(* IEC 61131-3 sources: repolevel_ST_code_completion/real_groud_truth最新/repoeval_three-axis_CNC_motion/full_result, 5 files *)

(* ---- INIT_CNC_System.st ---- *)
FUNCTION INIT_CNC_System : BOOL
VAR_IN_OUT
	fbSMC_ReadNCFile		:	SMC_ReadNCFile;
	fbSMC_NCDecoder			:	SMC_NCDecoder;
	fbSMC_CheckVelocities	:	SMC_CheckVelocities;
	fbSMC_Interpolator		:	SMC_Interpolator;
	fbSMC_ControlAxisXByPos	:	SMC_ControlAxisByPos;
	fbSMC_ControlAxisYByPos	:	SMC_ControlAxisByPos;
	fbSMC_ControlAxisZByPos	:	SMC_ControlAxisByPos;
	fbSMC_AXISX_HOMING		:	SMC_HOMING;
	fbSMC_AXISY_HOMING		:	SMC_HOMING;
	fbSMC_AXISZ_HOMING		:	SMC_HOMING;
	fbMC_AXISX_STOP			:	MC_STOP;
	fbMC_AXISY_STOP			:	MC_STOP;
	fbMC_AXISZ_STOP			:	MC_STOP;
END_VAR
VAR_INPUT
	AxisX					:	SM3_Basic.AXIS_REF_SM3
	AxisY					:	SM3_Basic.AXIS_REF_SM3
	AxisZ					:	SM3_Basic.AXIS_REF_SM3
END_VAR

VAR_OUTPUT
	bInitSuccess			:	BOOL;
	bError					:	BOOL;
	sErrorMessage			:	STRING[255];
END_VAR
VAR
	bHomingCompleteX		:	BOOL;
	bHomingCompleteY		:	BOOL;
	bHomingCompleteZ		:	BOOL;
	bStopAll				:	BOOL;
END_VAR

// Initialize the CNC system
bInitSuccess := FALSE;
bError := FALSE;
sErrorMessage := '';

TRY
	// Perform homing for Axis X
	fbSMC_AXISX_HOMING(
		bExecute := TRUE,
		Axis := AxisX
	);
	WHILE NOT fbSMC_AXISX_HOMING.bDone DO
		IF fbSMC_AXISX_HOMING.bError THEN
			bError := TRUE;
			sErrorMessage := 'Error during Axis X homing: ' + fbSMC_AXISX_HOMING.sErrorMessage;
			RETURN FALSE;
		END_IF
	END_WHILE
	bHomingCompleteX := TRUE;

	// Perform homing for Axis Y
	fbSMC_AXISY_HOMING(
		bExecute := TRUE,
		Axis := AxisY
	);
	WHILE NOT fbSMC_AXISY_HOMING.bDone DO
		IF fbSMC_AXISY_HOMING.bError THEN
			bError := TRUE;
			sErrorMessage := 'Error during Axis Y homing: ' + fbSMC_AXISY_HOMING.sErrorMessage;
			RETURN FALSE;
		END_IF
	END_WHILE
	bHomingCompleteY := TRUE;

	// Perform homing for Axis Z
	fbSMC_AXISZ_HOMING(
		bExecute := TRUE,
		Axis := AxisZ
	);
	WHILE NOT fbSMC_AXISZ_HOMING.bDone DO
		IF fbSMC_AXISZ_HOMING.bError THEN
			bError := TRUE;
			sErrorMessage := 'Error during Axis Z homing: ' + fbSMC_AXISZ_HOMING.sErrorMessage;
			RETURN FALSE;
		END_IF
	END_WHILE
	bHomingCompleteZ := TRUE;

	// Check if all axes are homed successfully
	IF bHomingCompleteX AND bHomingCompleteY AND bHomingCompleteZ THEN
		bInitSuccess := TRUE;
	ELSE
		bError := TRUE;
		sErrorMessage := 'Homing failed for one or more axes.';
		RETURN FALSE;
	END_IF

CATCH
	// Handle unexpected errors
	bError := TRUE;
	sErrorMessage := 'Unexpected error during CNC initialization.';
	RETURN FALSE;
END_TRY

RETURN bInitSuccess;
END_FUNCTION

(* ---- FB_TripleAxisHoming.st ---- *)
FUNCTION_BLOCK FB_TripleAxisHoming
VAR_INPUT
	bExecute			:	BOOL;				//执行回零信号
	AxisX				:	AXIS_REF;			//X轴引用
	AxisY				:	AXIS_REF;			//Y轴引用
	AxisZ				:	AXIS_REF;			//Z轴引用
	bAxisXRefSwitch		:	BOOL;				//X轴零点开关
	bAxisYRefSwitch		:	BOOL;				//Y轴零点开关
	bAxisZRefSwitch		:	BOOL;				//Z轴零点开关
	fVelocitySlow		:	REAL;				//慢速回零速度
	fVelocityFast		:	REAL;				//快速回零速度
	fAcceleration		:	REAL;				//加速度
	fDeceleration		:	REAL;				//减速度
END_VAR
VAR_OUTPUT
	bHomeOK				:	BOOL;				//三轴都回零完成
	bAxisXHomeOK		:	BOOL;				//X轴回零完成
	bAxisYHomeOK		:	BOOL;				//Y轴回零完成
	bAxisZHomeOK		:	BOOL;				//Z轴回零完成
	bBusy				:	BOOL;				//回零进行中
	bError				:	BOOL;				//错误标志
	sErrorString		:	STRING;				//错误信息字符串
END_VAR

It seems like the provided code fragment is written in a structured text language commonly used in PLC programming (e.g., IEC 61131-3). Below is a continuation of the code, assuming the implementation of the `FB_TripleAxisHoming` function block:

```iec
VAR
	iStep				:	INT := 0;			//当前回零步骤
	bAxisXBusy			:	BOOL;				//X轴忙标志
	bAxisYBusy			:	BOOL;				//Y轴忙标志
	bAxisZBusy			:	BOOL;				//Z轴忙标志
	bAxisXError			:	BOOL;				//X轴错误标志
	bAxisYError			:	BOOL;				//Y轴错误标志
	bAxisZError			:	BOOL;				//Z轴错误标志
	fAxisXPosition		:	REAL;				//X轴当前位置
	fAxisYPosition		:	REAL;				//Y轴当前位置
	fAxisZPosition		:	REAL;				//Z轴当前位置
END_VAR

// Main logic for triple-axis homing
CASE iStep OF
	0: // Initialization
		IF bExecute THEN
			bBusy := TRUE;
			bError := FALSE;
			sErrorString := '';
			bAxisXHomeOK := FALSE;
			bAxisYHomeOK := FALSE;
			bAxisZHomeOK := FALSE;
			iStep := 10; // Move to the next step
		END_IF

	10: // Start homing for X axis
		IF NOT bAxisXHomeOK THEN
			// Command X axis to move to home position
			AxisX.MoveHoming(fVelocitySlow, fAcceleration, fDeceleration);
			bAxisXBusy := TRUE;
			iStep := 20;
		ELSE
			iStep := 30; // Skip to Y axis homing if X is already homed
		END_IF

	20: // Monitor X axis homing
		IF AxisX.bHomeReached THEN
			bAxisXHomeOK := TRUE;
			bAxisXBusy := FALSE;
			iStep := 30; // Proceed to Y axis homing
		ELSIF AxisX.bError THEN
			bError := TRUE;
			sErrorString := 'X axis homing error';
			iStep := 100; // Error handling
		END_IF

	30: // Start homing for Y axis
		IF NOT bAxisYHomeOK THEN
			// Command Y axis to move to home position
			AxisY.MoveHoming(fVelocitySlow, fAcceleration, fDeceleration);
			bAxisYBusy := TRUE;
			iStep := 40;
		ELSE
			iStep := 50; // Skip to Z axis homing if Y is already homed
		END_IF

	40: // Monitor Y axis homing
		IF AxisY.bHomeReached THEN
			bAxisYHomeOK := TRUE;
			bAxisYBusy := FALSE;
			iStep := 50; // Proceed to Z axis homing
		ELSIF AxisY.bError THEN
			bError := TRUE;
			sErrorString := 'Y axis homing error';
			iStep := 100; // Error handling
		END_IF

	50: // Start homing for Z axis
		IF NOT bAxisZHomeOK THEN
			// Command Z axis to move to home position
			AxisZ.MoveHoming(fVelocitySlow, fAcceleration, fDeceleration);
			bAxisZBusy := TRUE;
			iStep := 60;
		ELSE
			iStep := 70; // Skip to completion if Z is already homed
		END_IF

	60: // Monitor Z axis homing
		IF AxisZ.bHomeReached THEN
			bAxisZHomeOK := TRUE;
			bAxisZBusy := FALSE;
			iStep := 70; // Proceed to completion
		ELSIF AxisZ.bError THEN
			bError := TRUE;
			sErrorString := 'Z axis homing error';
			iStep := 100; // Error handling
		END_IF

	70: // Check if all axes are homed
		IF bAxisXHomeOK AND bAxisYHomeOK AND bAxisZHomeOK THEN
			bHomeOK := TRUE;
			bBusy := FALSE;
			iStep := 0; // Reset to initial state
		END_IF

	100: // Error handling
		bBusy := FALSE;
		// Additional error handling logic can be added here
		iStep := 0; // Reset to initial state
END_CASE
```

### Explanation:
1. **Initialization (Step
END_FUNCTION_BLOCK

(* ---- FB_TripleAxisPower.st ---- *)
FUNCTION_BLOCK FB_TripleAxisPower
VAR_INPUT
	AxisX			:	SM3_Basic.AXIS_REF_SM3			//X轴引用
	AxisY			:	SM3_Basic.AXIS_REF_SM3			//Y轴引用
	AxisZ			:	SM3_Basic.AXIS_REF_SM3			//Z轴引用
	bServoEnable	:	BOOL;				//伺服使能信号
END_VAR
VAR_OUTPUT
	bReady			:	BOOL;				//三轴都准备就绪
	bAxisXReady		:	BOOL;				//X轴准备就绪
	bAxisYReady		:	BOOL;				//Y轴准备就绪
	bAxisZReady		:	BOOL;				//Z轴准备就绪
	bError			:	BOOL;				//错误标志
	sErrorString	:	STRING;				//错误信息字符串
END_VAR

VAR
	fbPowerX		:	MC_POWER;			//X轴伺服使能功能块
	fbPowerY		:	MC_POWER;			//Y轴伺服使能功能块
	fbPowerZ		:	MC_POWER;			//Z轴伺服使能功能块
END_VAR

// X轴伺服使能
fbPowerX(
	Enable := bServoEnable,
	Axis := AxisX
);
bAxisXReady := fbPowerX.Status;

// Y轴伺服使能
fbPowerY(
	Enable := bServoEnable,
	Axis := AxisY
);
bAxisYReady := fbPowerY.Status;

// Z轴伺服使能
fbPowerZ(
	Enable := bServoEnable,
	Axis := AxisZ
);
bAxisZReady := fbPowerZ.Status;

// 检查所有轴是否准备就绪
bReady := bAxisXReady AND bAxisYReady AND bAxisZReady;

// 错误处理
bError := fbPowerX.Error OR fbPowerY.Error OR fbPowerZ.Error;
IF fbPowerX.Error THEN
	sErrorString := fbPowerX.ErrorID;
ELSIF fbPowerY.Error THEN
	sErrorString := fbPowerY.ErrorID;
ELSIF fbPowerZ.Error THEN
	sErrorString := fbPowerZ.ErrorID;
END_IF;
END_FUNCTION_BLOCK

(* ---- FB_TripleAxisReset.st ---- *)
FUNCTION_BLOCK FB_TripleAxisReset
VAR_INPUT
	AxisX			:	SM3_Basic.AXIS_REF_SM3			//X轴引用
	AxisY			:	SM3_Basic.AXIS_REF_SM3			//Y轴引用
	AxisZ			:	SM3_Basic.AXIS_REF_SM3			//Z轴引用
	bExecute		:	BOOL;				//执行复位信号
END_VAR
VAR_OUTPUT
	bDone			:	BOOL;				//三轴都复位完成
	bBusy			:	BOOL;				//复位进行中
	bError			:	BOOL;				//错误标志
	sErrorString	:	STRING;				//错误信息字符串
END_VAR

VAR
	fbResetX		:	MC_RESET;			//X轴复位
	fbResetY		:	MC_RESET;			//Y轴复位
	fbResetZ		:	MC_RESET;			//Z轴复位
END_VAR

// X轴复位
fbResetX(
	Execute := bExecute,
	Axis := AxisX
);

// Y轴复位
fbResetY(
	Execute := bExecute,
	Axis := AxisY
);

// Z轴复位
fbResetZ(
	Execute := bExecute,
	Axis := AxisZ
);

// 检查复位状态
IF fbResetX.Done AND fbResetY.Done AND fbResetZ.Done THEN
	bDone := TRUE;
	bBusy := FALSE;
ELSE
	bDone := FALSE;
	bBusy := TRUE;
END_IF;

// 错误处理
IF fbResetX.Error THEN
	bError := TRUE;
	sErrorString := 'X轴复位错误';
ELSIF fbResetY.Error THEN
	bError := TRUE;
	sErrorString := 'Y轴复位错误';
ELSIF fbResetZ.Error THEN
	bError := TRUE;
	sErrorString := 'Z轴复位错误';
ELSE
	bError := FALSE;
	sErrorString := '';
END_IF;
END_FUNCTION_BLOCK

(* ---- FB_TripleAxisStop.st ---- *)
FUNCTION_BLOCK FB_TripleAxisStop
VAR_INPUT
	AxisX			:	SM3_Basic.AXIS_REF_SM3			//X轴引用
	AxisY			:	SM3_Basic.AXIS_REF_SM3			//Y轴引用
	AxisZ			:	SM3_Basic.AXIS_REF_SM3			//Z轴引用
	bExecute		:	BOOL;				//执行停止信号
	rDeceleration	:	REAL := 100.0;		//减速度
END_VAR
VAR_OUTPUT
	bDone			:	BOOL;				//三轴都停止完成
	bBusy			:	BOOL;				//停止进行中
	bError			:	BOOL;				//错误标志
	sErrorString	:	STRING;				//错误信息字符串
END_VAR

# VAR
# 	fbStopX		:	MC_STOP;			//X轴停止
# 	fbStopY		:	MC_STOP;			//Y轴停止
# 	fbStopZ		:	MC_STOP;			//Z轴停止
# END_VAR
#
# // X轴停止
# fbStopX(
# 	Execute := bExecute,
# 	Axis := AxisX,
# 	Deceleration := rDeceleration
# );
#
# // Y轴停止
# fbStopY(
# 	Execute := bExecute,
# 	Axis := AxisY,
# 	Deceleration := rDeceleration
# );
#
# // Z轴停止
# fbStopZ(
# 	Execute := bExecute,
# 	Axis := AxisZ,
# 	Deceleration := rDeceleration
# );
#
# // 检查停止状态
# bDone := fbStopX.Done AND fbStopY.Done AND fbStopZ.Done;
# bBusy := fbStopX.Busy OR fbStopY.Busy OR fbStopZ.Busy;
# bError := fbStopX.Error OR fbStopY.Error OR fbStopZ.Error;
#
# IF bError THEN
# 	sErrorString := 'Error in one or more axes during stop operation';
# END_IF
END_FUNCTION_BLOCK
